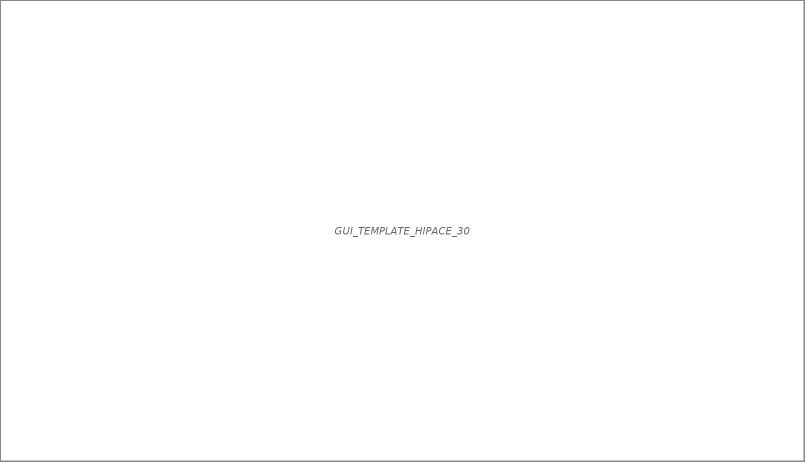
VISUALIZATION GUI_HIPACE_30_EVAC_PDS  // 805x462
    Frame (0,0 805x462)
        shows GUI_TEMPLATE_HIPACE_30(m_Instance := MAIN.evac_pds.tp, m_bEnable := MAIN.evac_pds.ctrl.bEnable_TP)
END_VISUALIZATION

(* stored: Version 1.1.0.1, ProductVersion 3.1.4024.9
   Visu GUI_HIPACE_30_EVAC_PDS: Id {be294070-3e0a-431a-8e68-578ee129e932} *)
